// TIA Portal V20 export
ORGANIZATION_BLOCK "MC_PreServo"   // OB67, LAD, PreServo
{ S7_Optimized_Access := 'TRUE' }
// stored: SetENOAutomatically false
   VAR_INPUT
      Initial_Call : Bool;
      PIP_Input : Bool;
      PIP_Output : Bool;
      IO_System : USInt;
      Event_Count : Int;
      Synchronous : Bool;
      CycleTime : UDInt;
   END_VAR
BEGIN

REGION Network 1
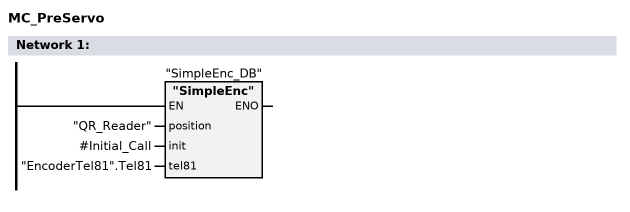
   RUNG wire#powerrail
      "SimpleEnc_DB"(position := "QR_Reader", init := #Initial_Call, tel81 := "EncoderTel81".Tel81)
   END_RUNG
   // the same network as SCL:
   "SimpleEnc_DB"(position := "QR_Reader", init := #Initial_Call, tel81 := "EncoderTel81".Tel81);   // "SimpleEnc"
END_REGION
END_ORGANIZATION_BLOCK
